TYPE ST_DischargeInCmd :
STRUCT
    bRun                : BOOL;
	bPause				: BOOL;
END_STRUCT
END_TYPE

(* stored: Version 1.1.0.1, ProductVersion 3.1.4024.16
   DUT ST_DischargeInCmd: Id {663ab9aa-da80-4713-a100-76597b8f569f} *)
